FUNCTION_BLOCK FB_LineRegulator EXTENDS MqttFramework.StateMachineLib.StateMachine
VAR_INPUT
END_VAR
VAR_OUTPUT
END_VAR
VAR
	fbTurntable : FB_Turntable;
	aRollerConveyors : ARRAY[1..3] OF FB_RollerConveyor;
END_VAR

Super^();

END_FUNCTION_BLOCK

(* stored: Version 1.1.0.1, ProductVersion 3.1.4024.0
   POU FB_LineRegulator: Id {ca3d4937-9986-4e8e-b7ee-5deb908a267b}, SpecialFunc None *)
